(* CoDeSys 2.3 export: _VALVE.EXP *)

(* Data type *)
TYPE _VALVE :
STRUCT
	xMode_AUTO : BOOL := FALSE; (* Активатия автоматического режима управления *)
	iValvePos : WORD; (* Текущее положение паравого клапана *)
	iSetPos : WORD; (* Заданное значение местоположения парового клапана *)
END_STRUCT
END_TYPE
